FUNCTION_BLOCK fbInheritanceLevel_5 EXTENDS fbInheritanceLevel_4
VAR
	{attribute addProperty Name "LEVEL 5"}
	level_5 : stAllTypes;		
END_VAR

METHOD Init : BOOL
VAR_INPUT
END_VAR
SUPER^.Init();
END_METHOD

END_FUNCTION_BLOCK

(* stored: Version 1.1.0.1, ProductVersion 3.1.4024.4
   POU fbInheritanceLevel_5: Id {74807b99-3731-41e6-9f64-0e44d94b184c}, SpecialFunc None
   Method Init: Id {582b02c7-0761-4a1c-9aa6-e674b19e672f} *)
